{attribute 'linkalways'} 
{attribute 'no_explicit_call' := 'This FB is a CLASS and must be accessed using methods or properties'}
{attribute 'enable_dynamic_creation'}
FUNCTION_BLOCK Node_F_VN_SetPixel EXTENDS VisionNode
VAR
    ipSrcImage : _ITcVnImage;
    aValue : _TcVnVector4_LREAL;
    nX : _UDINT(0);
    nY : _UDINT(0);
    hrPrev : _HRESULT(S_OK);
	hresult : _HRESULT(S_OK);
END_VAR

METHOD PUBLIC  Clone : I_Node
VAR
	pNode : POINTER TO Node_F_VN_SetPixel;
END_VAR
pNode := __NEW(Node_F_VN_SetPixel);
Clone := pNode^;
END_METHOD

METHOD FB_init : BOOL
VAR_INPUT
	bInitRetains : BOOL; // if TRUE, the retain variables are initialized (warm start / cold start)
	bInCopyCode : BOOL;  // if TRUE, the instance afterwards gets moved into the copy code (online change)
END_VAR
AddInput('ipSrcImage', ipSrcImage);
AddInput('aValue', aValue);
AddParameter('nX', nX);
AddParameter('nY', nY);
AddInput('hrPrev', hrPrev);
AddOutput('hresult',hresult);
END_METHOD

METHOD PROTECTED OnExecute
hresult.Value := F_VN_SetPixel(
    ipSrcImage := ipSrcImage.Value,
    aValue := aValue.Value,
    nX := nX.Value,
    nY := nY.Value,
	hrPrev:= hrPrev.Value);
END_METHOD

METHOD PUBLIC PreExecutionCheck
VAR_INPUT
	Check : I_PreExecutionChecks;
END_VAR
Check.IsTrue(ipSrcImage.IsValid, 'ipSrcImage must contain an image');
END_METHOD

END_FUNCTION_BLOCK

(* stored: Version 1.1.0.1, ProductVersion 3.1.4024.13
   POU Node_F_VN_SetPixel: Id {f3584eeb-3ae7-02ce-03ff-3e3c02ebf12b}, SpecialFunc None
   Folder Constructor: Id {1c67a358-b625-0f85-2d8d-54abf644b70d}
   Method Clone: Id {d948b31c-3e7b-0b23-173b-2a5f328709c6}
   Method FB_init: Id {3b863202-720f-05eb-398b-5ba6add29f7b}
   Method OnExecute: Id {f2bf4c54-d0f8-06fd-1be5-87cb8c6e6c3c}
   Method PreExecutionCheck: Id {0138ba2b-058d-09cd-3600-78be5155c952} *)
